// TIA Portal V20 export
VAR_GLOBAL   // PLC tag table "LKinCtrl_HMI_Diagnostics_Messages"
END_VAR
VAR_GLOBAL CONSTANT   // user constants
   LKINCTRL_MESSAGE_INDEX_OVERVIEW_RESET_SUCCESSFULL : Int := 2000;   // Info: 1-6999, Warning: 7000-7999, Error: 8000-
   LKINCTRL_MESSAGE_INDEX_OVERVIEW_ERROR_DURING_RESET : Int := 10000;   // Info: 1-6999, Warning: 7000-7999, Error: 8000-
END_VAR
